Staubli VAL3: S7telegram_T.dtx

public num H[18]
public num DATA[240]
